FUNCTION_BLOCK GearMover EXTENDS FB_Mover IMPLEMENTS IGearMover
VAR_INPUT
	XtsTrack : IXtsTrack;
	StateMachine : IPmlStateMachine;
END_VAR
VAR_OUTPUT
END_VAR
VAR
	moverSequence : GearMoverSequence;
	bInit : BOOL;
	CurrentLimit AT%Q* : INT;
	Mode AT%Q* : UINT;
	axesGear	: GearInCA;
	isMasterAxis: BOOL;
	MoverToGearTo: UDINT := 1;
END_VAR
VAR_IN_OUT
	MoverArray : ARRAY[*] OF IGearMover;
END_VAR

IF NOT bInit THEN
	_trackLength := XtsTrack.TrackLength;
	IF THIS^._axis.NcToPlc.AxisId <> 0 THEN
		IF (THIS^._axis.NcToPlc.AxisId MOD 2)<>1 THEN
			Mode.8 := TRUE;
			isMasterAxis := TRUE;
		ELSE
			isMasterAxis := FALSE;
			MoverToGearTo := THIS^.AxisRef.NcToPlc.AxisId + 1;
		END_IF
		bInit := TRUE;
	END_IF
END_IF

IF isMasterAxis THEN
	IF (_axis.NcToPlc.ModuloActPos > 3400 OR _axis.NcToPlc.ModuloActPos < 300)  THEN
		CurrentLimit := 1000;
	ELSE
		CurrentLimit := 2000;
	END_IF
ELSE
	CurrentLimit := 12000;
END_IF

SUPER^();
axesGear(_MasterAxis := MoverArray[MoverToGearTo].AxisRef, _SlaveAxis := THIS^.AxisRef);
moverSequence(ThisMover := THIS^,
				XtsTrack := XtsTrack,
				StateMachine := StateMachine,
				MoverArray := MoverArray);

METHOD PUBLIC Gear : BOOL
VAR_INPUT
	MasterPosition : MC_LREAL;
	SlavePosition : MC_LREAL;
END_VAR
IF NOT axesGear.Busy THEN
		axesGear.Sync(MasterPosition := MasterPosition, SlavePosition := SlavePosition);
		Gear := TRUE;
END_IF
END_METHOD

METHOD inGear : BOOL
VAR_INPUT
END_VAR
inGear := axesGear.gearInCA.InSync;
END_METHOD

METHOD isMaster : BOOL
VAR_INPUT
END_VAR
isMaster := isMasterAxis;
END_METHOD

METHOD masterAxis : UDINT
VAR_INPUT
END_VAR
masterAxis := MoverToGearTo;
END_METHOD

END_FUNCTION_BLOCK

(* stored: Version 1.1.0.1, ProductVersion 3.1.4024.11
   POU GearMover: Id {0fe93f55-b780-4d7c-972c-ecf14934b0c1}, SpecialFunc None
   Method Gear: Id {7681a46f-476d-4db2-a300-5813fc91eee6}
   Method inGear: Id {6de601b6-d26a-4174-b6fd-96c961e5fce9}
   Method isMaster: Id {80b75d0a-70e8-4b4a-88fe-d22b2582fcfd}
   Method masterAxis: Id {580ce28e-8614-4edd-b50d-08a75fd63cf2} *)
